Yaskawa INFORM job: TEST.JBI

/JOB
//NAME TEST
//POS
///NPOS 3,3,3,0,0,0
///TOOL 0
///POSTYPE ROBOT
///RECTAN
///RCONF 0,0,0,0,1,0,0,0,0,0,0,0,0,0,0,0,0,0,0,0,0,0,0,0
C00000=2166.047,-134.022,-1141.160,-7.3080,-53.9216,4.1035
C00001=2166.047,-134.022,-1141.160,-7.3080,-53.9216,4.1035
C00002=2166.047,-134.022,-1141.160,-7.3080,-53.9216,4.1035
///RCONF 0,0,0,0,0,0,0,0,0,0,0,0,0,0,0,0,0,0,0,0,0,0,0,0
BC00000=385.118,3798.148,919.771
BC00001=385.118,3798.148,919.771
BC00002=385.118,3798.148,919.771
///POSTYPE PULSE
///PULSE
EC00000=1,1
EC00001=1,1
EC00002=1,1
//INST
///DATE 2024/01/29 18:05
///ATTR SC,RW,RJ
////FRAME ROBOT
///GROUP1 RB1,BS1
///GROUP2 ST1
NOP
SMOVL C00000 BC00000 V=11.0  +MOVJ EC00000
SMOVL C00001 BC00001 V=11.7  +MOVJ EC00001 VJ=0.78
SMOVL C00002 BC00002 V=11.7  +MOVJ EC00002 VJ=0.78
END
